// TIA Portal V18 export
// export: Created 2026-06-08T05:50:11Z, ExportSetting WithDefaults
PlcWatchTable "WT_Test_Import_DB_Schema"
  PlcWatchTableEntry ""DB_PLC1_Send_To_PLC2_DB".CmdSeq"
